// TIA Portal V16 export
// export: Created 2021-11-12T13:31:04.2917412Z, ExportSetting WithDefaults, DisplayName Totally Integrated Automation Portal, DisplayVersion V16 Update 3, DisplayName TIA Portal Version Control Interface, DisplayVersion V16 Update 2, DisplayName TIA Portal Openness, DisplayVersion V16 Update 3, DisplayName SINAMICS Startdrive Advanced, DisplayVersion V16 Update 5, DisplayName SINAMICS Startdrive G130, G150, S120, S150, SINAMICS MV, S210, DisplayVersion V16 Update 5, DisplayName SINAMICS Startdrive G110M, G120, G120C, G120D, G120P, G115D, DisplayVersion V16 Update 5, DisplayName STEP 7 Professional, DisplayVersion V16 Update 3, DisplayName STEP 7 Safety, DisplayVersion V16, DisplayName WinCC UA Professional, DisplayVersion V16 Update 3
DATA_BLOCK "Sfty_InterfaceStd"   // DB6
{ S7_Optimized_Access := 'TRUE'; DB_Accessible_From_OPC_UA := 'FALSE' }
VERSION : 0.1
// stored: AutoNumber true, DBAccessibleFromOPCUA false, IsOnlyStoredInLoadMemory false, IsRetainMemResEnabled false, IsWriteProtectedInAS false, MemoryReserve 100
   VAR
      ACK { S7_SetPoint := 'True'} : "UDT_AckSafety";   // Acknowledgement groups
      "100RU01-QQ01_In" { S7_SetPoint := 'True'} : "UDT_LockOut";   // Inputs from safety program
      "100RU01-QQ02_In" { S7_SetPoint := 'True'} : "UDT_LockOut";   // Inputs from safety program
      "100RU01-QQ03_In" { S7_SetPoint := 'True'} : "UDT_LockOut";   // Inputs from safety program
      "100RU01-QQ04_In" { S7_SetPoint := 'True'} : "UDT_LockOut";   // Inputs from safety program
      "100RU01-QQ05_In" { S7_SetPoint := 'True'} : "UDT_LockOut";   // Inputs from safety program
      "100RU01-QQ06_In" { S7_SetPoint := 'True'} : "UDT_LockOut";   // Inputs from safety program
      "100RU01-QQ07_In" { S7_SetPoint := 'True'} : "UDT_LockOut";   // Inputs from safety program
      "100RU01-QQ08_In" { S7_SetPoint := 'True'} : "UDT_LockOut";   // Inputs from safety program
      "200RU01-QQ01_In" { S7_SetPoint := 'True'} : "UDT_LockOut";   // Inputs from safety program
      "200RU01-QQ02_In" { S7_SetPoint := 'True'} : "UDT_LockOut";   // Inputs from safety program
      "200RU01-QQ03_In" { S7_SetPoint := 'True'} : "UDT_LockOut";   // Inputs from safety program
      "200RU01-QQ04_In" { S7_SetPoint := 'True'} : "UDT_LockOut";   // Inputs from safety program
      "200RU01-QQ05_In" { S7_SetPoint := 'True'} : "UDT_LockOut";   // Inputs from safety program
      "100RU01-QQ01_Out" { S7_SetPoint := 'True'} : "UDT_LockIn";   // Outputs to safety program
      "100RU01-QQ02_Out" { S7_SetPoint := 'True'} : "UDT_LockIn";   // Outputs to safety program
      "100RU01-QQ03_Out" { S7_SetPoint := 'True'} : "UDT_LockIn";   // Outputs to safety program
      "100RU01-QQ04_Out" { S7_SetPoint := 'True'} : "UDT_LockIn";   // Outputs to safety program
      "100RU01-QQ05_Out" { S7_SetPoint := 'True'} : "UDT_LockIn";   // Outputs to safety program
      "100RU01-QQ06_Out" { S7_SetPoint := 'True'} : "UDT_LockIn";   // Outputs to safety program
      "100RU01-QQ07_Out" { S7_SetPoint := 'True'} : "UDT_LockIn";   // Outputs to safety program
      "100RU01-QQ08_Out" { S7_SetPoint := 'True'} : "UDT_LockIn";   // Outputs to safety program
      "200RU01-QQ01_Out" { S7_SetPoint := 'True'} : "UDT_LockIn";   // Outputs to safety program
      "200RU01-QQ02_Out" { S7_SetPoint := 'True'} : "UDT_LockIn";   // Outputs to safety program
      "200RU01-QQ03_Out" { S7_SetPoint := 'True'} : "UDT_LockIn";   // Outputs to safety program
      "200RU01-QQ04_Out" { S7_SetPoint := 'True'} : "UDT_LockIn";   // Outputs to safety program
      "200RU01-QQ05_Out" { S7_SetPoint := 'True'} : "UDT_LockIn";   // Outputs to safety program
   END_VAR
BEGIN
END_DATA_BLOCK
